Staubli VAL3: AA_Chessie.pjx

--- AA_Chessie.pjx ---
Parameters version=s7.9 stackSize=5000 millimeterUnit=true
Program file=CasesNoires.pgx
Program file=Data_acqu.pgx
Program file=DeplacementInit.pgx
Program file=Deplacementpion.pgx
Program file=Pionperdu.pgx
Program file=start.pgx
Program file=stop.pgx
Program file=TestPositionCal.pgx
Data file=AA_Chessie.dtx

--- AA_Chessie.dtx ---
frame fFrame = {x=374.8, y=3.07, z=-517.036829, rx=-180, fatherId=world[0]}
jointRx jCaseNoire = {j1=-5.017205, j2=92.568227, j3=85.506286, j4=-5.02125, j5=92.334481, j6=182.995856}
jointRx jDepart = {j1=20.811233, j2=126.617326, j3=-10.855704, j5=64.238378, j6=-69.188767}
jointRx jInitial
jointRx jStart = {j1=-4.35, j2=22.39, j3=131, j5=25.77, j6=50.65}
mdesc mDeplacement = {accel=200}
mdesc mDepose = {accel=25, vel=50}
mdesc mPrise = {accel=25, vel=50}
num nTESTSIO[66]
num nX = 4
num nY = 9
num nData[10]
num ni = 32
pointRx pCaseNoire[33]
  [0] = {x=374.8, y=3.07, z=-495.75, rx=-180, shoulder=lefty, elbow=epositive, wrist=wpositive, fatherId=world[0]}
  [1] = {x=430.4, y=3.07, z=-495.75, rx=-180, shoulder=lefty, elbow=epositive, wrist=wpositive, fatherId=world[0]}
  [2] = {x=486, y=3.07, z=-495.75, rx=-180, shoulder=lefty, elbow=epositive, wrist=wpositive, fatherId=world[0]}
  [3] = {x=541.6, y=3.07, z=-495.75, rx=-180, shoulder=lefty, elbow=epositive, wrist=wpositive, fatherId=world[0]}
  [4] = {x=402.6, y=30.87, z=-495.75, rx=-180, shoulder=lefty, elbow=epositive, wrist=wpositive, fatherId=world[0]}
  [5] = {x=458.2, y=30.87, z=-495.75, rx=-180, shoulder=lefty, elbow=epositive, wrist=wpositive, fatherId=world[0]}
  [6] = {x=513.8, y=30.87, z=-495.75, rx=-180, shoulder=lefty, elbow=epositive, wrist=wpositive, fatherId=world[0]}
  [7] = {x=569.4, y=30.87, z=-495.75, rx=-180, shoulder=lefty, elbow=epositive, wrist=wpositive, fatherId=world[0]}
  [8] = {x=374.8, y=58.67, z=-495.75, rx=-180, shoulder=lefty, elbow=epositive, wrist=wpositive, fatherId=world[0]}
  [9] = {x=430.4, y=58.67, z=-495.75, rx=-180, shoulder=lefty, elbow=epositive, wrist=wpositive, fatherId=world[0]}
  [10] = {x=486, y=58.67, z=-495.75, rx=-180, shoulder=lefty, elbow=epositive, wrist=wpositive, fatherId=world[0]}
  [11] = {x=541.6, y=58.67, z=-495.75, rx=-180, shoulder=lefty, elbow=epositive, wrist=wpositive, fatherId=world[0]}
  [12] = {x=402.6, y=86.47, z=-495.75, rx=-180, shoulder=lefty, elbow=epositive, wrist=wpositive, fatherId=world[0]}
  [13] = {x=458.2, y=86.47, z=-495.75, rx=-180, shoulder=lefty, elbow=epositive, wrist=wpositive, fatherId=world[0]}
  [14] = {x=513.8, y=86.47, z=-495.75, rx=-180, shoulder=lefty, elbow=epositive, wrist=wpositive, fatherId=world[0]}
  [15] = {x=569.4, y=86.47, z=-495.75, rx=-180, shoulder=lefty, elbow=epositive, wrist=wpositive, fatherId=world[0]}
  [16] = {x=374.8, y=114.27, z=-495.75, rx=-180, shoulder=lefty, elbow=epositive, wrist=wpositive, fatherId=world[0]}
  [17] = {x=430.4, y=114.27, z=-495.75, rx=-180, shoulder=lefty, elbow=epositive, wrist=wpositive, fatherId=world[0]}
  [18] = {x=486, y=114.27, z=-495.75, rx=-180, shoulder=lefty, elbow=epositive, wrist=wpositive, fatherId=world[0]}
  [19] = {x=541.6, y=114.27, z=-495.75, rx=-180, shoulder=lefty, elbow=epositive, wrist=wpositive, fatherId=world[0]}
  [20] = {x=402.6, y=142.07, z=-495.75, rx=-180, shoulder=lefty, elbow=epositive, wrist=wpositive, fatherId=world[0]}
  [21] = {x=458.2, y=142.07, z=-495.75, rx=-180, shoulder=lefty, elbow=epositive, wrist=wpositive, fatherId=world[0]}
  [22] = {x=513.8, y=142.07, z=-495.75, rx=-180, shoulder=lefty, elbow=epositive, wrist=wpositive, fatherId=world[0]}
  [23] = {x=569.4, y=142.07, z=-495.75, rx=-180, shoulder=lefty, elbow=epositive, wrist=wpositive, fatherId=world[0]}
  [24] = {x=374.8, y=169.87, z=-495.75, rx=-180, shoulder=lefty, elbow=epositive, wrist=wpositive, fatherId=world[0]}
  [25] = {x=430.4, y=169.87, z=-495.75, rx=-180, shoulder=lefty, elbow=epositive, wrist=wpositive, fatherId=world[0]}
  [26] = {x=486, y=169.87, z=-495.75, rx=-180, shoulder=lefty, elbow=epositive, wrist=wpositive, fatherId=world[0]}
  [27] = {x=541.6, y=169.87, z=-495.75, rx=-180, shoulder=lefty, elbow=epositive, wrist=wpositive, fatherId=world[0]}
  [28] = {x=402.6, y=197.67, z=-495.75, rx=-180, shoulder=lefty, elbow=epositive, wrist=wpositive, fatherId=world[0]}
  [29] = {x=458.2, y=197.67, z=-495.75, rx=-180, shoulder=lefty, elbow=epositive, wrist=wpositive, fatherId=world[0]}
  [30] = {x=513.8, y=197.67, z=-495.75, rx=-180, shoulder=lefty, elbow=epositive, wrist=wpositive, fatherId=world[0]}
  [31] = {x=569.4, y=197.67, z=-495.75, rx=-180, shoulder=lefty, elbow=epositive, wrist=wpositive, fatherId=world[0]}
  [32] = {fatherId=world[0]}
pointRx pPieceMangees[26]
  [0] = {x=374.8, y=-97.99178, z=-500.37, rx=-180, shoulder=lefty, elbow=epositive, wrist=wpositive, fatherId=world[0]}
  [1] = {x=394.8, y=-97.99178, z=-500.37, rx=-180, shoulder=lefty, elbow=epositive, wrist=wpositive, fatherId=world[0]}
  [2] = {x=414.8, y=-97.99178, z=-500.37, rx=-180, shoulder=lefty, elbow=epositive, wrist=wpositive, fatherId=world[0]}
  [3] = {x=434.8, y=-97.99178, z=-500.37, rx=-180, shoulder=lefty, elbow=epositive, wrist=wpositive, fatherId=world[0]}
  [4] = {x=454.8, y=-97.99178, z=-500.37, rx=-180, shoulder=lefty, elbow=epositive, wrist=wpositive, fatherId=world[0]}
  [5] = {x=474.8, y=-97.99178, z=-500.37, rx=-180, shoulder=lefty, elbow=epositive, wrist=wpositive, fatherId=world[0]}
  [6] = {x=374.8, y=-117.99178, z=-500.37, rx=-180, shoulder=lefty, elbow=epositive, wrist=wpositive, fatherId=world[0]}
  [7] = {x=394.8, y=-117.99178, z=-500.37, rx=-180, shoulder=lefty, elbow=epositive, wrist=wpositive, fatherId=world[0]}
  [8] = {x=414.8, y=-117.99178, z=-500.37, rx=-180, shoulder=lefty, elbow=epositive, wrist=wpositive, fatherId=world[0]}
  [9] = {x=434.8, y=-117.99178, z=-500.37, rx=-180, shoulder=lefty, elbow=epositive, wrist=wpositive, fatherId=world[0]}
  [10] = {x=454.8, y=-117.99178, z=-500.37, rx=-180, shoulder=lefty, elbow=epositive, wrist=wpositive, fatherId=world[0]}
  [11] = {x=474.8, y=-117.99178, z=-500.37, rx=-180, shoulder=lefty, elbow=epositive, wrist=wpositive, fatherId=world[0]}
  [12] = {x=374.8, y=-137.99178, z=-500.37, rx=-180, shoulder=lefty, elbow=epositive, wrist=wpositive, fatherId=world[0]}
  [13] = {x=394.8, y=-137.99178, z=-500.37, rx=-180, shoulder=lefty, elbow=epositive, wrist=wpositive, fatherId=world[0]}
  [14] = {x=414.8, y=-137.99178, z=-500.37, rx=-180, shoulder=lefty, elbow=epositive, wrist=wpositive, fatherId=world[0]}
  [15] = {x=434.8, y=-137.99178, z=-500.37, rx=-180, shoulder=lefty, elbow=epositive, wrist=wpositive, fatherId=world[0]}
  [16] = {x=454.8, y=-137.99178, z=-500.37, rx=-180, shoulder=lefty, elbow=epositive, wrist=wpositive, fatherId=world[0]}
  [17] = {x=474.8, y=-137.99178, z=-500.37, rx=-180, shoulder=lefty, elbow=epositive, wrist=wpositive, fatherId=world[0]}
  [18] = {x=374.8, y=-157.99178, z=-500.37, rx=-180, shoulder=lefty, elbow=epositive, wrist=wpositive, fatherId=world[0]}
  [19] = {x=394.8, y=-157.99178, z=-500.37, rx=-180, shoulder=lefty, elbow=epositive, wrist=wpositive, fatherId=world[0]}
  [20] = {x=414.8, y=-157.99178, z=-500.37, rx=-180, shoulder=lefty, elbow=epositive, wrist=wpositive, fatherId=world[0]}
  [21] = {x=434.8, y=-157.99178, z=-500.37, rx=-180, shoulder=lefty, elbow=epositive, wrist=wpositive, fatherId=world[0]}
  [22] = {x=454.8, y=-157.99178, z=-500.37, rx=-180, shoulder=lefty, elbow=epositive, wrist=wpositive, fatherId=world[0]}
  [23] = {x=474.8, y=-157.99178, z=-500.37, rx=-180, shoulder=lefty, elbow=epositive, wrist=wpositive, fatherId=world[0]}
  [24] = {x=374.8, y=-177.99178, z=-500.37, rx=-180, shoulder=lefty, elbow=epositive, wrist=wpositive, fatherId=world[0]}
  [25] = {x=394.8, y=-177.99178, z=-500.37, rx=-180, shoulder=lefty, elbow=epositive, wrist=wpositive, fatherId=world[0]}
pointRx pTable = {fatherId=fFrame[0]}
public sio sData = {link=Socket\staubli_server}
tool tTool = {x=63.134763, y=38.954373, z=16.017439, rx=-90.869915, ry=61.402378, rz=90.763801, fatherId=flange[0], ioLink=valve1}
trsf trAppro = {z=-40}
string sString[2]
  [0] = "nTESTIO"
  [1] = "nTESTIO"
num i
num nb
num TEST[10]
num Compteur_perdu

--- start.pgx ---
public program start()
begin
  // Position des cases
  //   28   29  30  31             ligne 8
  //     ....                      ...
  //  8   9  10  11                ligne 3
  //    4   5   6   7              ligne 2
  //  0   1   2   3                ligne 1
  //pCase[0] = case O en bas à gauche du plateau

  //se met en position 0
  //  call DeplacementInit()

  //Deplacementpion(X,Y) -> deplacement du pion de X vers Y
  //  call Deplacementpion(0,4)

  //call TestPositionCal()

  call DeplacementInit()
  call Data_acqu()

  if TEST[2]==0
    call Deplacementpion(TEST[0],TEST[1])

  else
    call Deplacementpion(TEST[0],TEST[1])
    call Pionperdu(TEST[2],Compteur_perdu)
    Compteur_perdu=Compteur_perdu+1
  endIf
end

--- CasesNoires.pgx ---
public program CasesNoires()
begin


  // Position des cases
  //   28   29  30  31             ligne 8
  //     ....                      ...
  //  8   9  10  11                ligne 3
  //    4   5   6   7              ligne 2
  //  0   1   2   3                ligne 1

  //pCase[0] = case O en bas à gauche du plateau

  //variable pour numeroter les cases
  ni=0

  for nY=1 to 8
    for nX=0 to 3

      //ligne case impair
      if nY%2==1
        pCaseNoire[ni]=compose(pCaseNoire[0],fFrame,{55.6*nX,-27.8*(nY-1),0,0,0,0})
        //pCaseNoire[ni]= pCaseNoire[0] + 55.6*nX + 27.8 * (nY - 1)

        //ligne case pair
      else
        pCaseNoire[ni]=compose(pCaseNoire[0],fFrame,{27.8*(nX+1)+27.8*nX,-27.8*(nY-1),0,0,0,0})
        //pCaseNoire[ni]= pCaseNoire[0] + 27.8*(nX+1) + 27.8 * (nY - 1)
      endIf

      ni=ni+1

    endFor
  endFor


end

--- Data_acqu.pgx ---
program Data_acqu()
begin

  sioCtrl(sData, "port", 5000)
  sioCtrl(sData, "clients", 1)
  //On choisit un caractère de fin de ligne
  sioCtrl(sData, "endOfString", 33)
  logMsg("------------ Sio Initialise")
  // ---- Programme pour lire une trsf ----
  nb=0
  i=0

  while(nb<24)
    //sioGet renvoie le nombre de caractère lue sur la liaison
    //elle convertit en ASCII la valeur reçue et la stock dans nTESTIO dans notre cas
    nb=sioGet(sData, nTESTSIO[i])
    sString=toString("",nTESTSIO[i])
    logMsg("donnee recu")
    logMsg(sString)
    delay(0.5)
    if(nb>0)
      i=i+nb
    else
      // Erreur de communication
      return
    endIf
  endWhile
  logMsg("fin du train de donnée")
  logMsg("début de la conversion")
  if(fromBinary(nTESTSIO, 24, "8.0l", TEST) != 3)
    // Données altérées
    logMsg("données altérées")
    return
  else
    logMsg("conversion réussie")
    sString=toString("",TEST[0])
    logMsg(sString)
    sString=toString("",TEST[1])
    logMsg(sString)
    logMsg("deplacement")
    //call Deplacementpion(1,TEST)
  endIf

end

--- DeplacementInit.pgx ---
program DeplacementInit()
begin
  movej(jInitial,tTool,mDeplacement)
end

--- Deplacementpion.pgx ---
public program Deplacementpion(num x_nPointDepart (dimensions=1), num x_nPointArrivee (dimensions=1))
begin
  //met à jour position des cases noires
  call CasesNoires()


  //Deplacementpion(X,Y) -> deplacement du pion de X vers Y


  //Deplacement vers le pion en X
  movej(appro(pCaseNoire[x_nPointDepart],trAppro),tTool,mDeplacement)

  //s'approche et prend le pion en X
  close(tTool)
  movel(pCaseNoire[x_nPointDepart],tTool,mPrise)
  open(tTool)

  movel(appro(pCaseNoire[x_nPointDepart],trAppro),tTool,mDeplacement)

  //Deplacement vers Y puis approche vers Y
  movej(appro(pCaseNoire[x_nPointArrivee],trAppro),tTool,mDeplacement)
  movel(pCaseNoire[x_nPointArrivee],tTool,mPrise)

  //lache la piece et remonte
  close(tTool)
  movel(appro(pCaseNoire[x_nPointArrivee],trAppro),tTool,mDeplacement)


end

--- Pionperdu.pgx ---
program Pionperdu(num x_nPionperdu (dimensions=1), num x_nPionjete (dimensions=1))
begin
  //met à jour position des cases noires

  //Deplacementpion(X,Y) -> deplacement du pion de X vers Y


  //Deplacement vers le pion en X
  movej(appro(pCaseNoire[x_nPionperdu],trAppro),tTool,mDeplacement)

  //s'approche et prend le pion en X
  close(tTool)
  movel(pCaseNoire[x_nPionperdu],tTool,mPrise)
  open(tTool)

  movel(appro(pCaseNoire[x_nPionperdu],trAppro),tTool,mDeplacement)

  //Deplacement vers Y puis approche vers Y
  movej(appro(pPieceMangees[x_nPionjete],trAppro),tTool,mDeplacement)
  movel(pPieceMangees[x_nPionjete],tTool,mPrise)

  //lache la piece et remonte
  close(tTool)
  movel(appro(pPieceMangees[x_nPionjete],trAppro),tTool,mDeplacement)


end

--- TestPositionCal.pgx ---
program TestPositionCal()
begin
  call DeplacementInit()

  call Deplacementpion(9,13)
  call Deplacementpion(22,18)

  call Deplacementpion(13,22)
  call Pionperdu(18,0)

  call Deplacementpion(26,19)
  call Pionperdu(22,1)

  call DeplacementInit()

end
